// SIMATIC S7-200 project (STEP 7-Micro/WIN), CPU 224XP REL 02.01

ORGANIZATION_BLOCK MAIN:OB1
TITLE=程序注释
BEGIN
Network 2
AB=    VB135, 2
AB=    VB101, 35
AB=    VB112, 36
Network 3
AB=    VB135, 3
AB=    VB101, 35
AB=    VB126, 36
Network 5
AB<>   SMB186, 0
RCV    VB100, 0
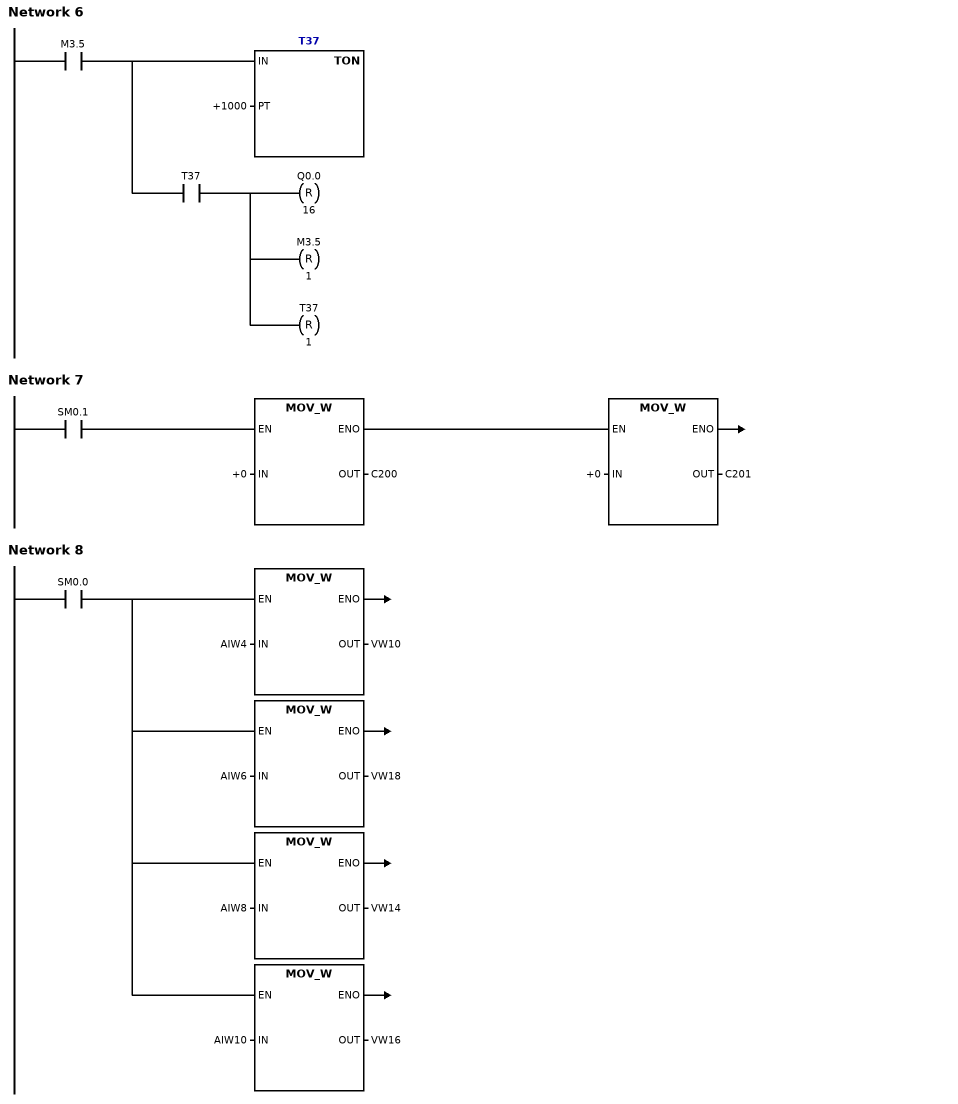
Network 6
LD     M3.5
TON    T37, +1000
A      T37
R      Q0.0, 16
R      M3.5, 1
R      T37, 1
Network 7
LD     SM0.1
MOVW   +0, C200
AENO
MOVW   +0, C201
Network 8
LD     SM0.0
MOVW   AIW4, VW10
MOVW   AIW6, VW18
MOVW   AIW8, VW14
MOVW   AIW10, VW16
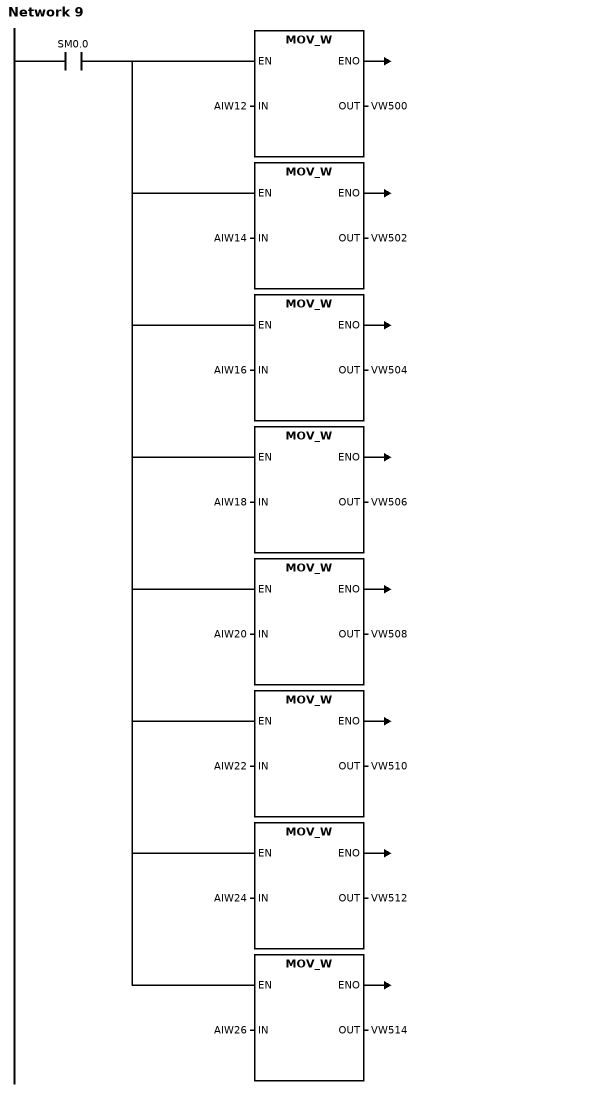
Network 9
LD     SM0.0
MOVW   AIW12, VW500
MOVW   AIW14, VW502
MOVW   AIW16, VW504
MOVW   AIW18, VW506
MOVW   AIW20, VW508
MOVW   AIW22, VW510
MOVW   AIW24, VW512
MOVW   AIW26, VW514
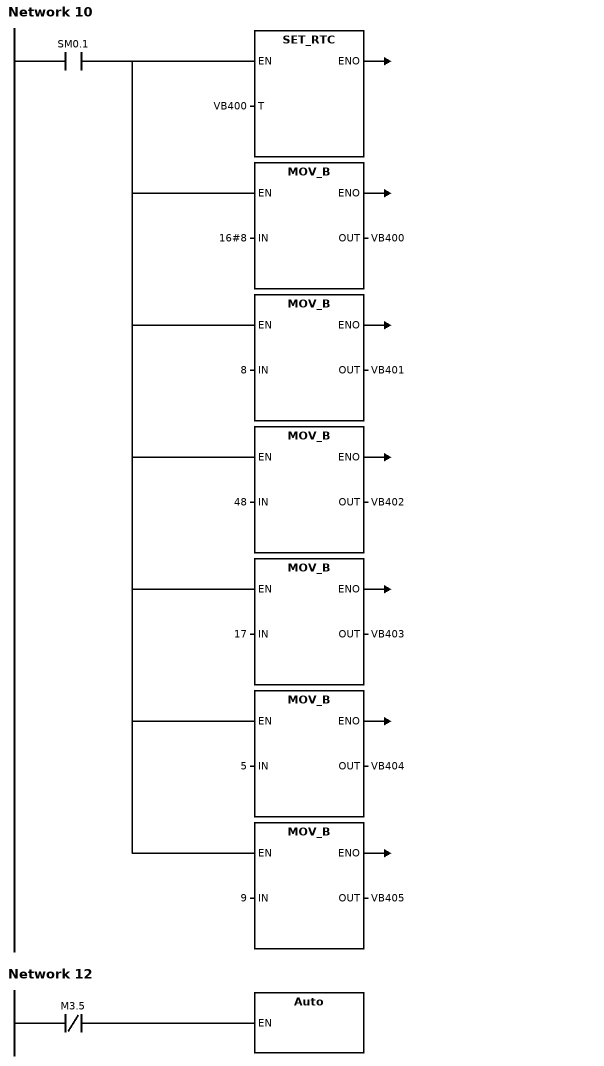
Network 10
LD     SM0.1
TODW   VB400
MOVB   16#8, VB400
MOVB   8, VB401
MOVB   48, VB402
MOVB   17, VB403
MOVB   5, VB404
MOVB   9, VB405
Network 11
LDN    I4.7
Network 12
LDN    M3.5
CALL   Auto:SBR4
Network 13
AB=    VB135, 1
AB=    VB101, 35
AB=    VB106, 36
Network 14
AB=    VB135, 5
AB=    VB101, 35
AB=    VB106, 36
S      M18.0, 1
Network 15
AB=    VB135, 6
AB=    VB101, 35
AB=    VB106, 36
S      M18.1, 1
END_ORGANIZATION_BLOCK

SUBROUTINE_BLOCK Auto:SBR4
TITLE=
BEGIN
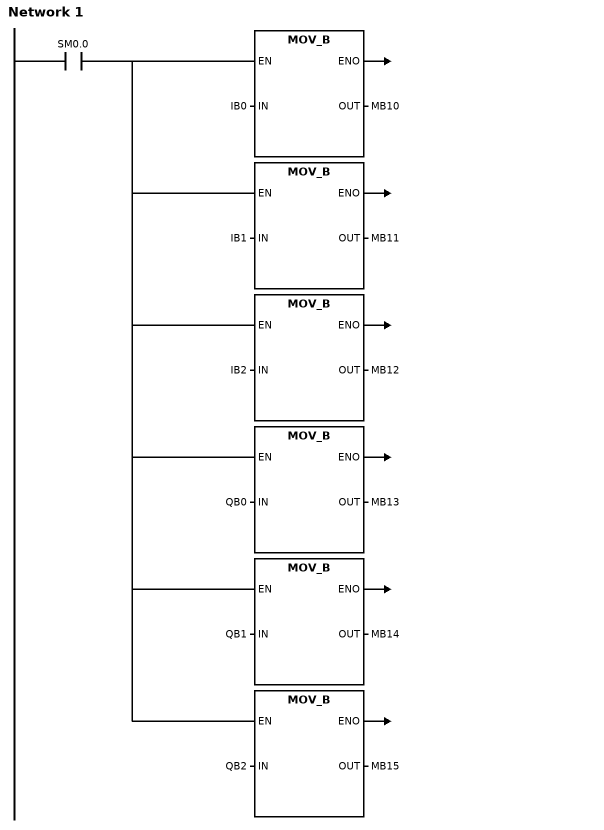
Network 1
LD     SM0.0
MOVB   IB0, MB10
MOVB   IB1, MB11
MOVB   IB2, MB12
MOVB   QB0, MB13
MOVB   QB1, MB14
MOVB   QB2, MB15
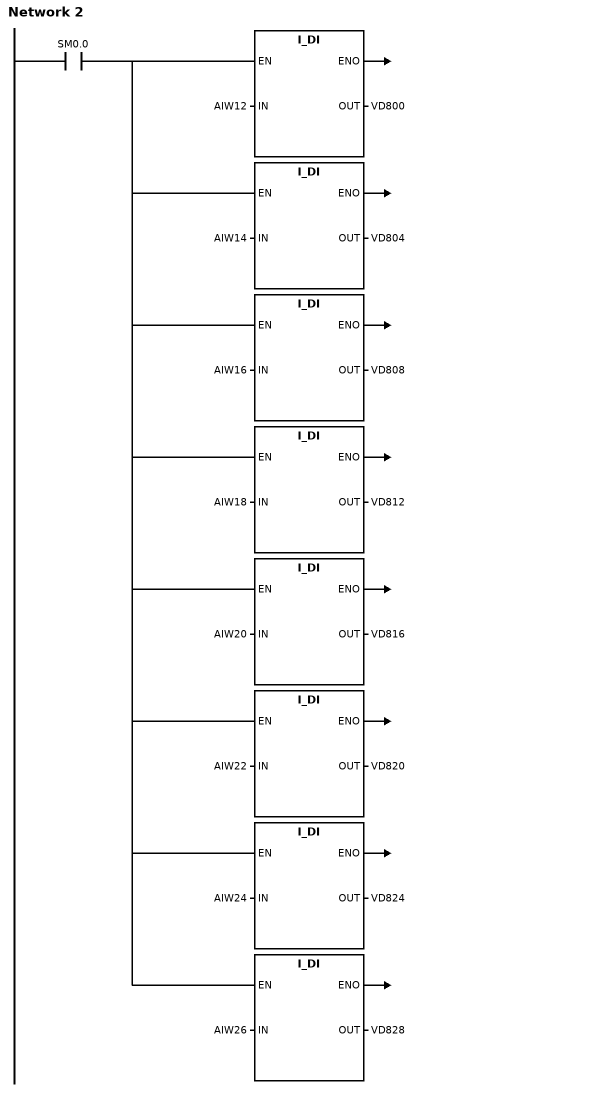
Network 2
LD     SM0.0
ITD    AIW12, VD800
ITD    AIW14, VD804
ITD    AIW16, VD808
ITD    AIW18, VD812
ITD    AIW20, VD816
ITD    AIW22, VD820
ITD    AIW24, VD824
ITD    AIW26, VD828
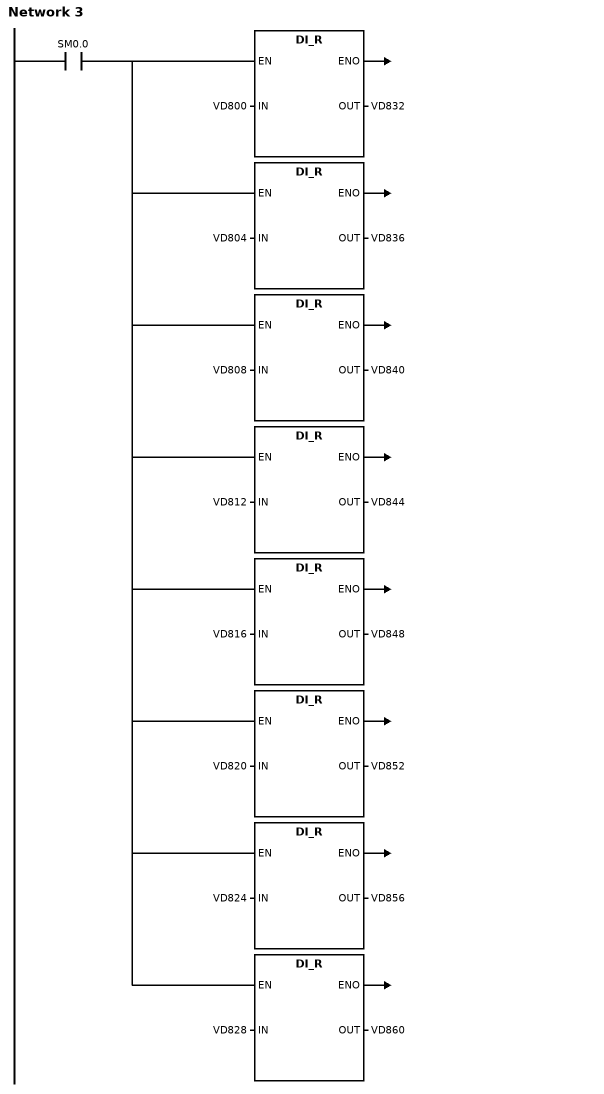
Network 3
LD     SM0.0
DTR    VD800, VD832
DTR    VD804, VD836
DTR    VD808, VD840
DTR    VD812, VD844
DTR    VD816, VD848
DTR    VD820, VD852
DTR    VD824, VD856
DTR    VD828, VD860
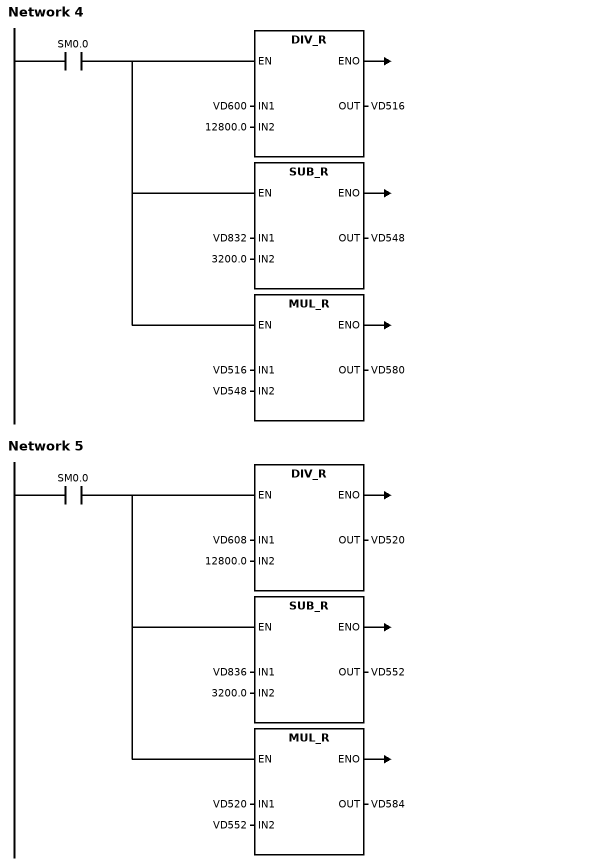
Network 4
LD     SM0.0
MOVR   VD600, VD516
/R     12800.0, VD516
MOVR   VD832, VD548
-R     3200.0, VD548
MOVR   VD516, VD580
*R     VD548, VD580
Network 5
LD     SM0.0
MOVR   VD608, VD520
/R     12800.0, VD520
MOVR   VD836, VD552
-R     3200.0, VD552
MOVR   VD520, VD584
*R     VD552, VD584
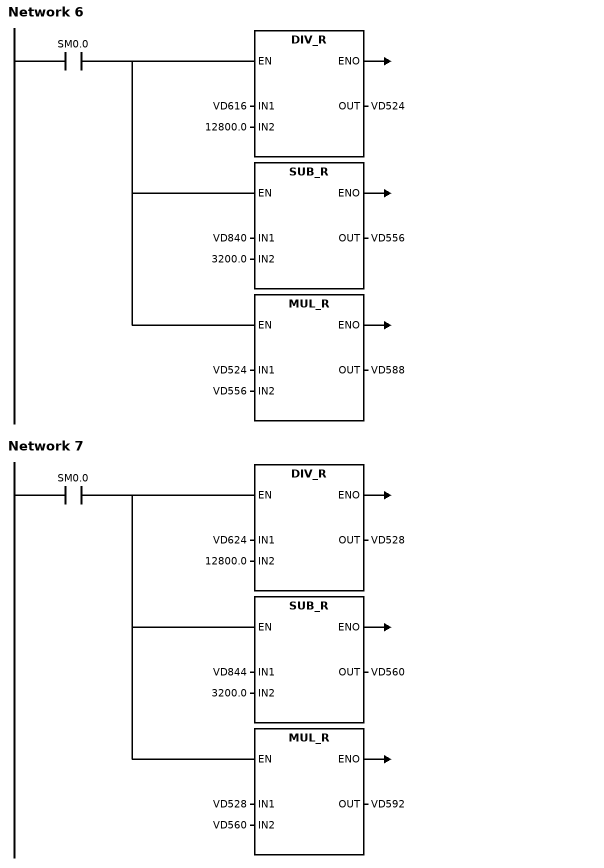
Network 6
LD     SM0.0
MOVR   VD616, VD524
/R     12800.0, VD524
MOVR   VD840, VD556
-R     3200.0, VD556
MOVR   VD524, VD588
*R     VD556, VD588
Network 7
LD     SM0.0
MOVR   VD624, VD528
/R     12800.0, VD528
MOVR   VD844, VD560
-R     3200.0, VD560
MOVR   VD528, VD592
*R     VD560, VD592
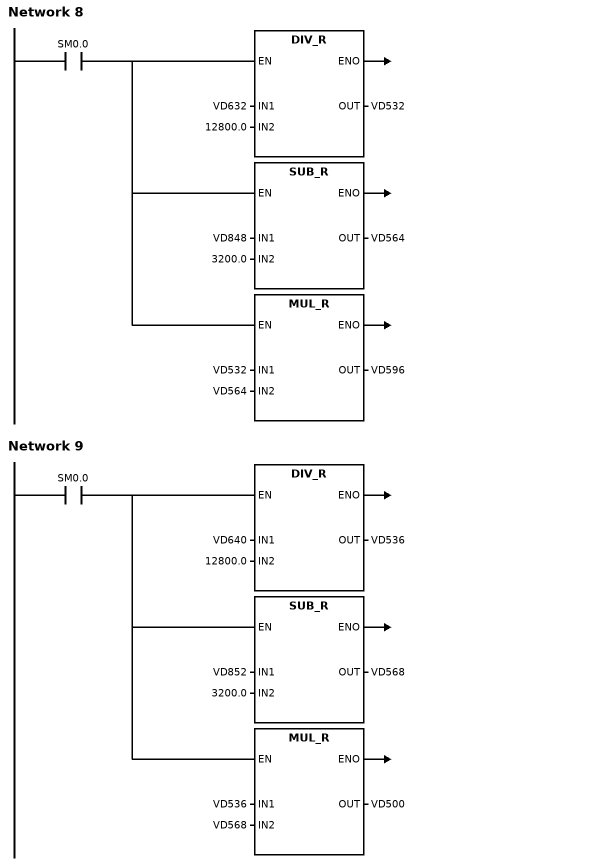
Network 8
LD     SM0.0
MOVR   VD632, VD532
/R     12800.0, VD532
MOVR   VD848, VD564
-R     3200.0, VD564
MOVR   VD532, VD596
*R     VD564, VD596
Network 9
LD     SM0.0
MOVR   VD640, VD536
/R     12800.0, VD536
MOVR   VD852, VD568
-R     3200.0, VD568
MOVR   VD536, VD500
*R     VD568, VD500
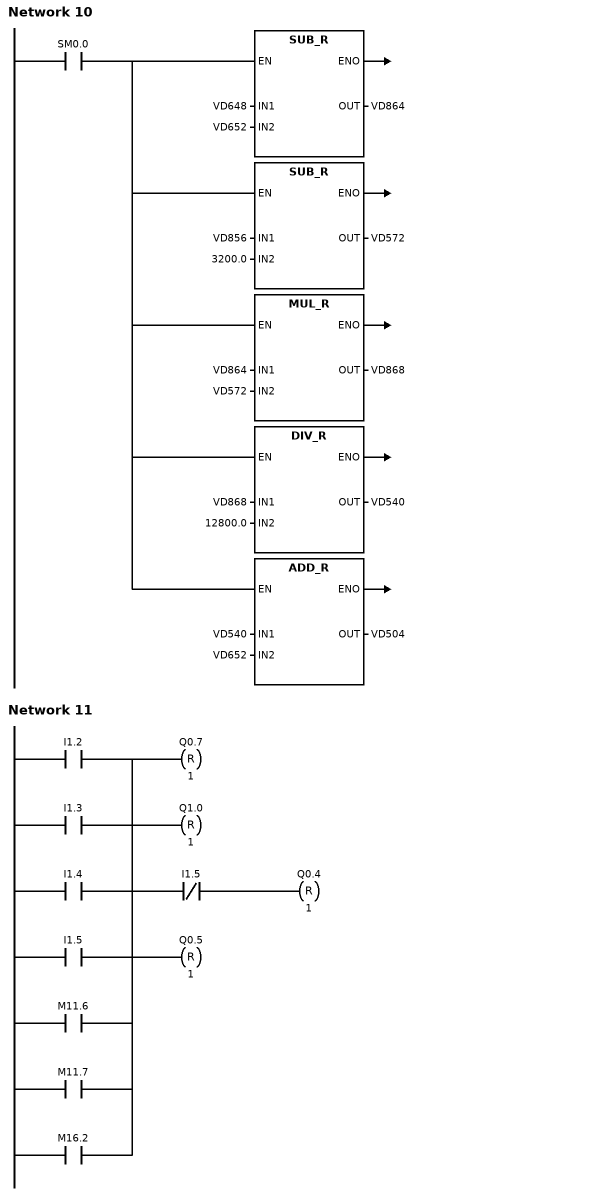
Network 10
LD     SM0.0
MOVR   VD648, VD864
-R     VD652, VD864
MOVR   VD856, VD572
-R     3200.0, VD572
MOVR   VD864, VD868
*R     VD572, VD868
MOVR   VD868, VD540
/R     12800.0, VD540
MOVR   VD540, VD504
+R     VD652, VD504
Network 11
LD     I1.2
O      I1.3
O      I1.4
O      I1.5
O      M11.6
O      M11.7
O      M16.2
LPS
R      Q0.7, 1
R      Q1.0, 1
AN     I1.5
R      Q0.4, 1
LPP
R      Q0.5, 1
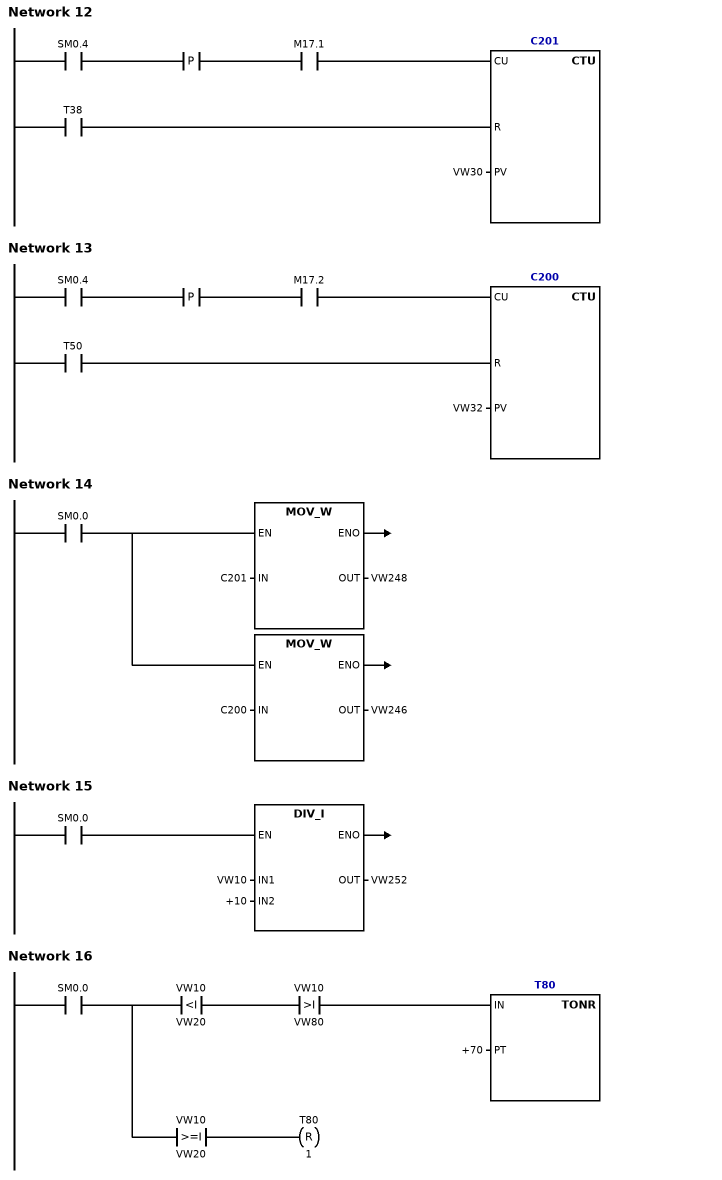
Network 12
LD     SM0.4
EU
A      M17.1
LD     T38
CTU    C201, VW30
Network 13
LD     SM0.4
EU
A      M17.2
LD     T50
CTU    C200, VW32
Network 14
LD     SM0.0
MOVW   C201, VW248
MOVW   C200, VW246
Network 15
LD     SM0.0
MOVW   VW10, VW252
/I     +10, VW252
Network 16
LD     SM0.0
LPS
AW<    VW10, VW20
AW>    VW10, VW80
TONR   T80, +70
LPP
AW>=   VW10, VW20
R      T80, 1
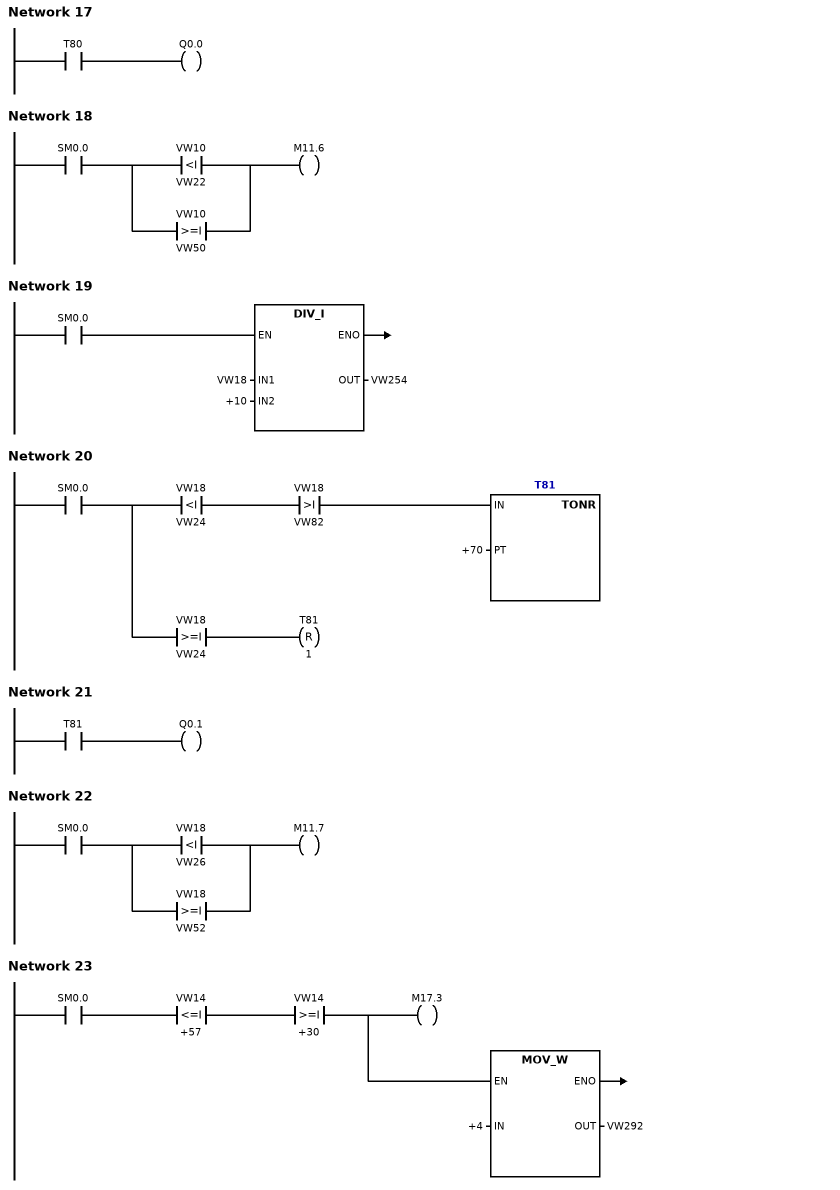
Network 17
LD     T80
=      Q0.0
Network 18
LD     SM0.0
LDW<   VW10, VW22
OW>=   VW10, VW50
ALD
=      M11.6
Network 19
LD     SM0.0
MOVW   VW18, VW254
/I     +10, VW254
Network 20
LD     SM0.0
LPS
AW<    VW18, VW24
AW>    VW18, VW82
TONR   T81, +70
LPP
AW>=   VW18, VW24
R      T81, 1
Network 21
LD     T81
=      Q0.1
Network 22
LD     SM0.0
LDW<   VW18, VW26
OW>=   VW18, VW52
ALD
=      M11.7
Network 23
LD     SM0.0
AW<=   VW14, +57
AW>=   VW14, +30
=      M17.3
MOVW   +4, VW292
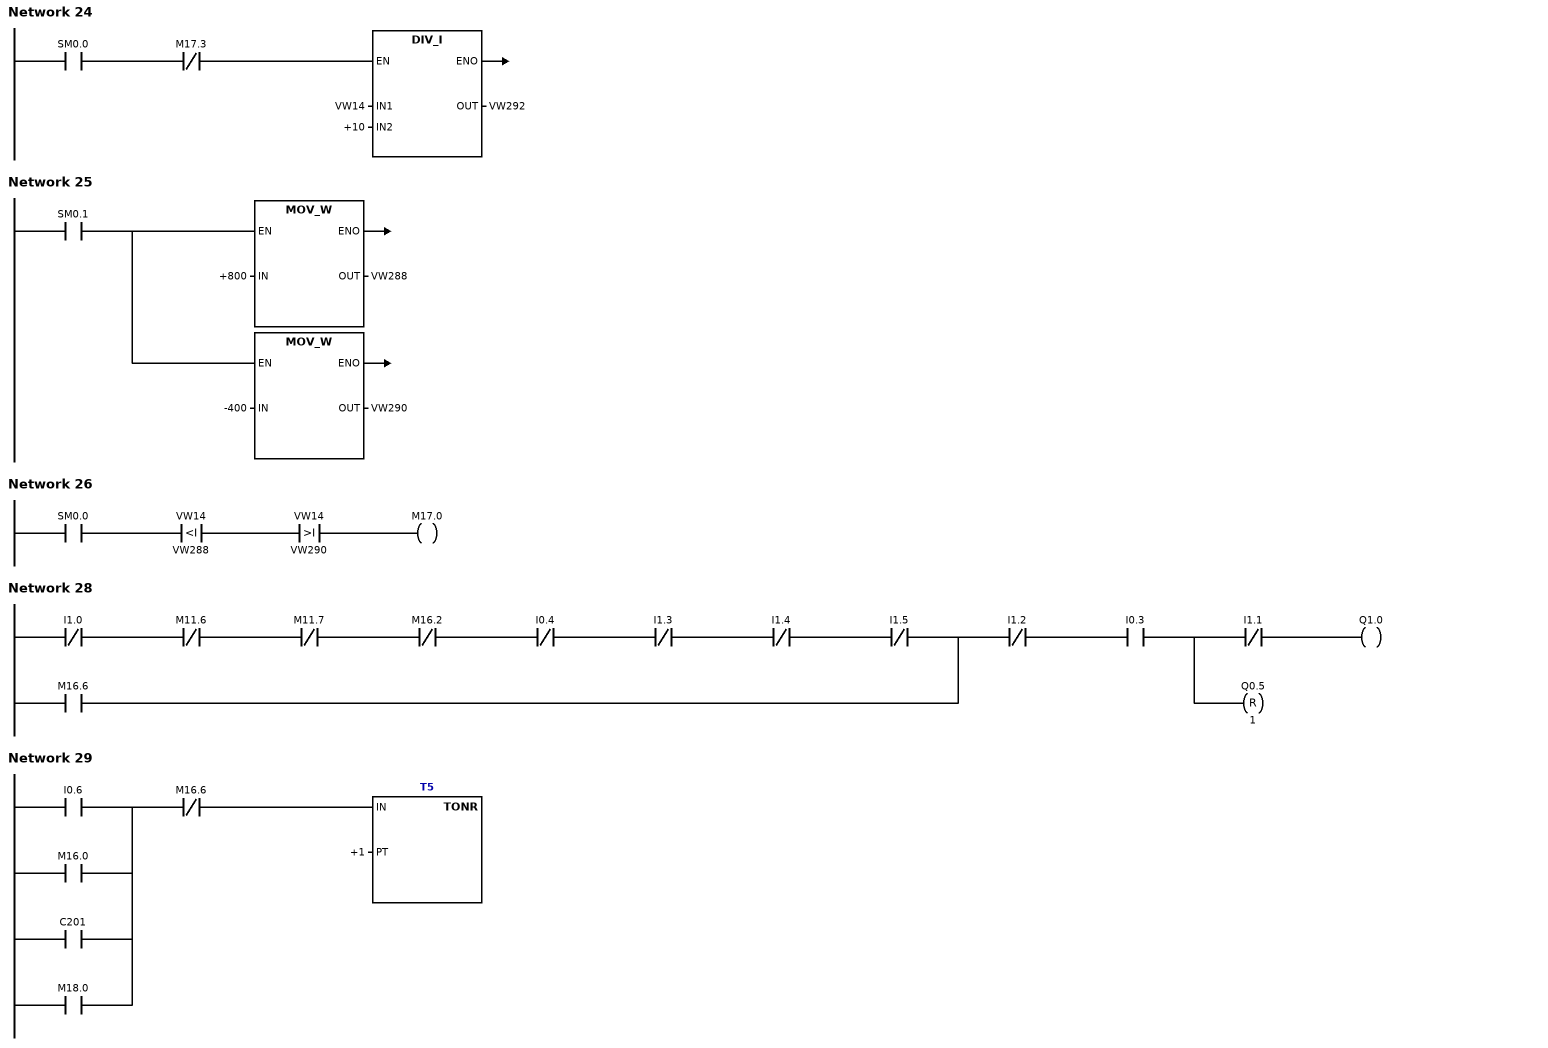
Network 24
LD     SM0.0
AN     M17.3
MOVW   VW14, VW292
/I     +10, VW292
Network 25
LD     SM0.1
MOVW   +800, VW288
MOVW   -400, VW290
Network 26
LD     SM0.0
AW<    VW14, VW288
AW>    VW14, VW290
=      M17.0
Network 28
LDN    I1.0
AN     M11.6
AN     M11.7
AN     M16.2
AN     I0.4
AN     I1.3
AN     I1.4
AN     I1.5
O      M16.6
AN     I1.2
A      I0.3
LPS
AN     I1.1
=      Q1.0
LPP
R      Q0.5, 1
Network 29
LD     I0.6
O      M16.0
O      C201
O      M18.0
AN     M16.6
TONR   T5, +1
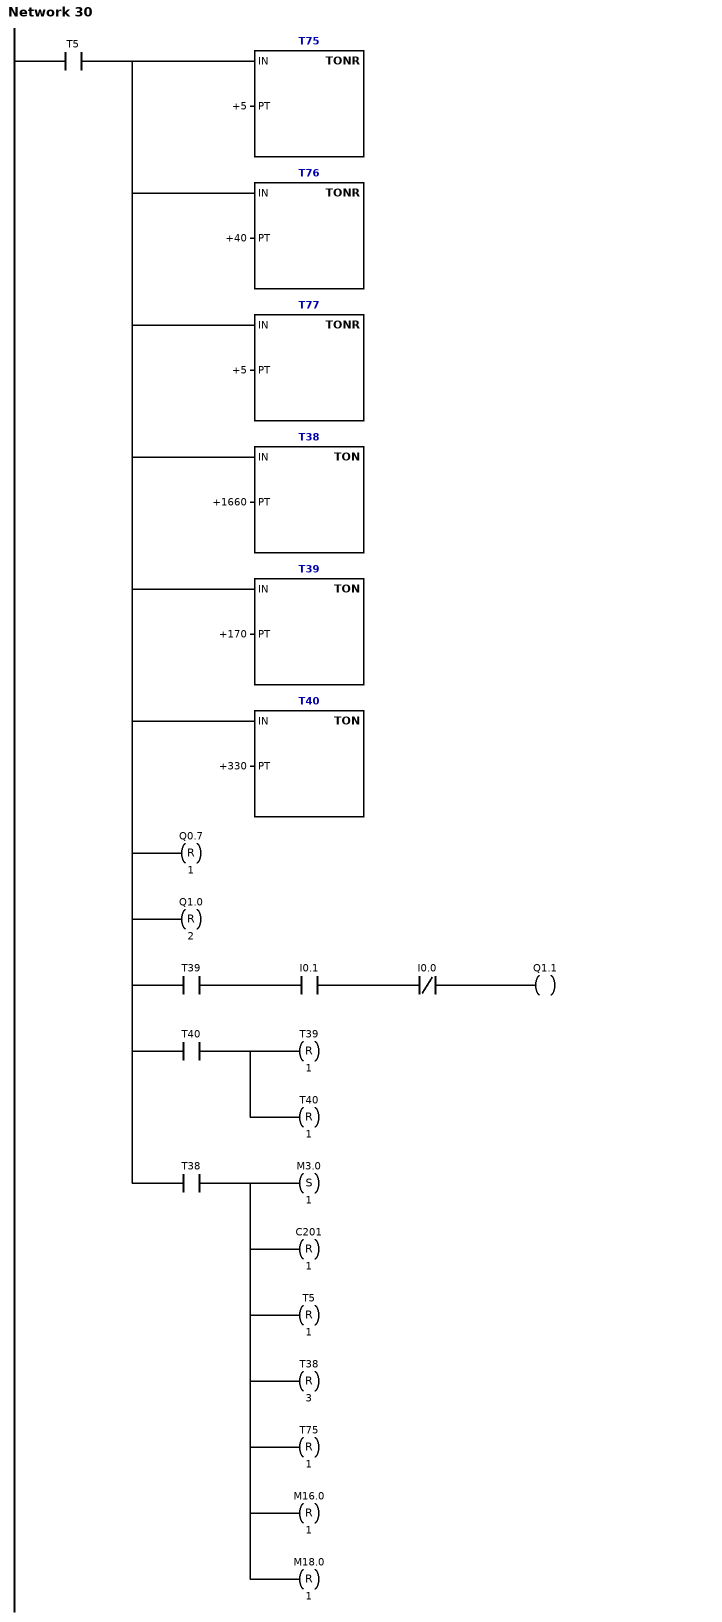
Network 30
LD     T5
LPS
TONR   T75, +5
TONR   T76, +40
TONR   T77, +5
TON    T38, +1660
TON    T39, +170
TON    T40, +330
R      Q0.7, 1
R      Q1.0, 2
A      T39
A      I0.1
AN     I0.0
=      Q1.1
LRD
A      T40
R      T39, 1
R      T40, 1
LPP
A      T38
S      M3.0, 1
R      C201, 1
R      T5, 1
R      T38, 3
R      T75, 1
R      M16.0, 1
R      M18.0, 1
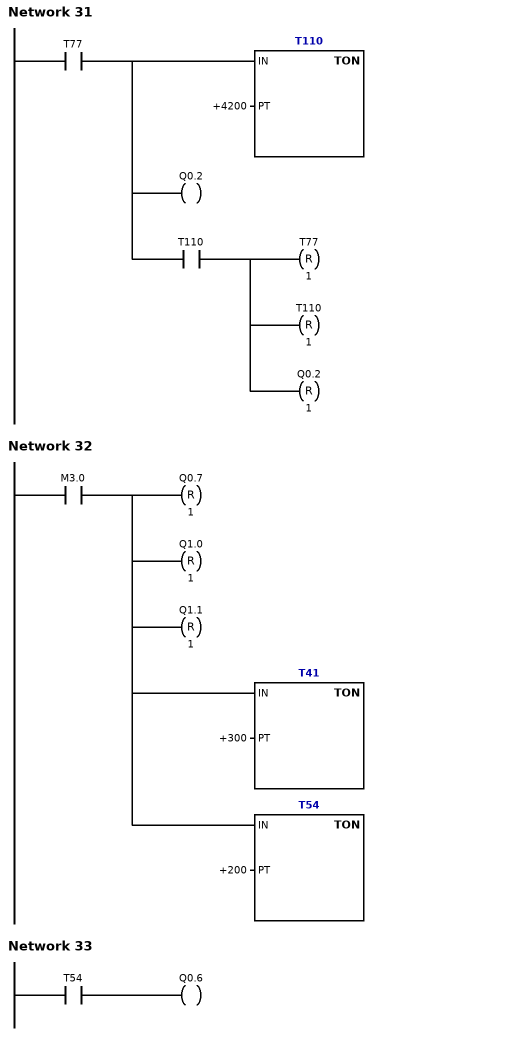
Network 31
LD     T77
TON    T110, +4200
=      Q0.2
A      T110
R      T77, 1
R      T110, 1
R      Q0.2, 1
Network 32
LD     M3.0
R      Q0.7, 1
R      Q1.0, 1
R      Q1.1, 1
TON    T41, +300
TON    T54, +200
Network 33
LD     T54
=      Q0.6
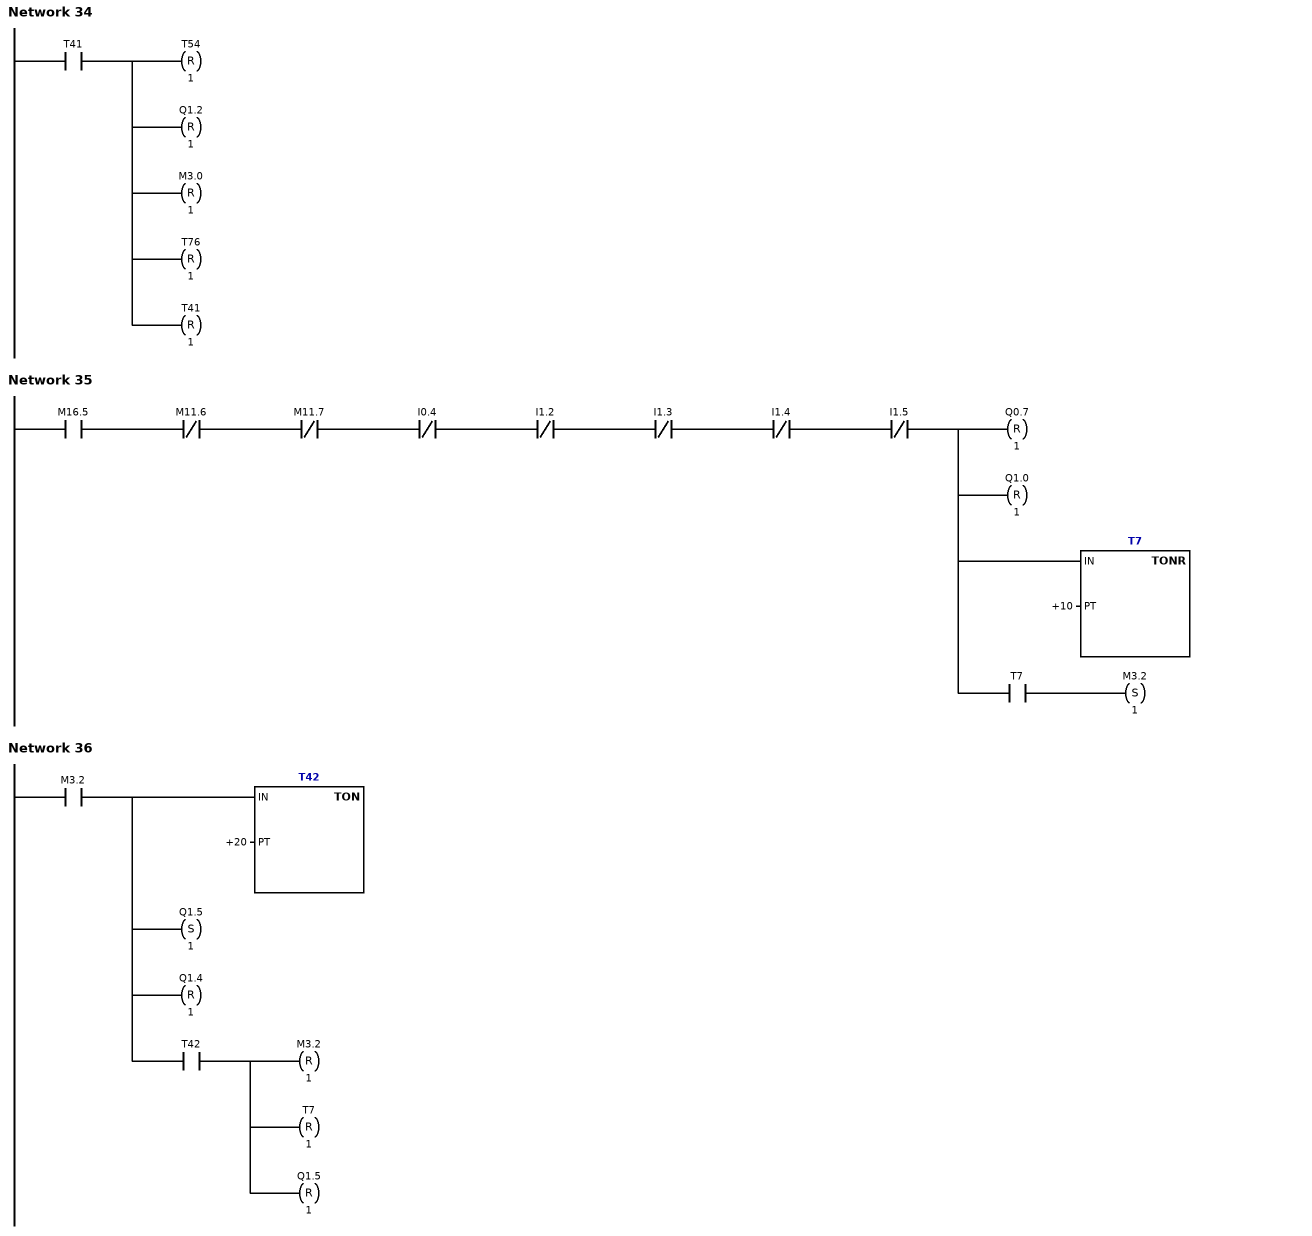
Network 34
LD     T41
R      T54, 1
R      Q1.2, 1
R      M3.0, 1
R      T76, 1
R      T41, 1
Network 35
LD     M16.5
AN     M11.6
AN     M11.7
AN     I0.4
AN     I1.2
AN     I1.3
AN     I1.4
AN     I1.5
R      Q0.7, 1
R      Q1.0, 1
TONR   T7, +10
A      T7
S      M3.2, 1
Network 36
LD     M3.2
TON    T42, +20
S      Q1.5, 1
R      Q1.4, 1
A      T42
R      M3.2, 1
R      T7, 1
R      Q1.5, 1
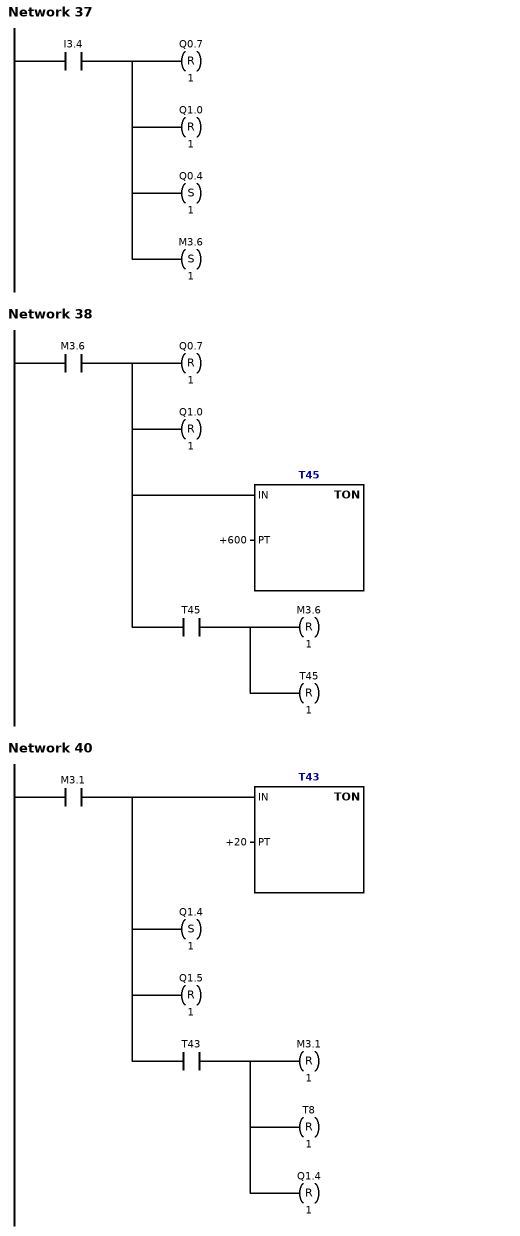
Network 37
LD     I3.4
R      Q0.7, 1
R      Q1.0, 1
S      Q0.4, 1
S      M3.6, 1
Network 38
LD     M3.6
R      Q0.7, 1
R      Q1.0, 1
TON    T45, +600
A      T45
R      M3.6, 1
R      T45, 1
Network 39
AN     M11.6
AN     M11.7
AN     I1.0
AN     I1.2
AN     I1.3
AN     I1.4
AN     I1.5
R      Q0.7, 1
R      Q1.0, 1
TONR   T8, +10
A      T8
S      M3.1, 1
Network 40
LD     M3.1
TON    T43, +20
S      Q1.4, 1
R      Q1.5, 1
A      T43
R      M3.1, 1
R      T8, 1
R      Q1.4, 1
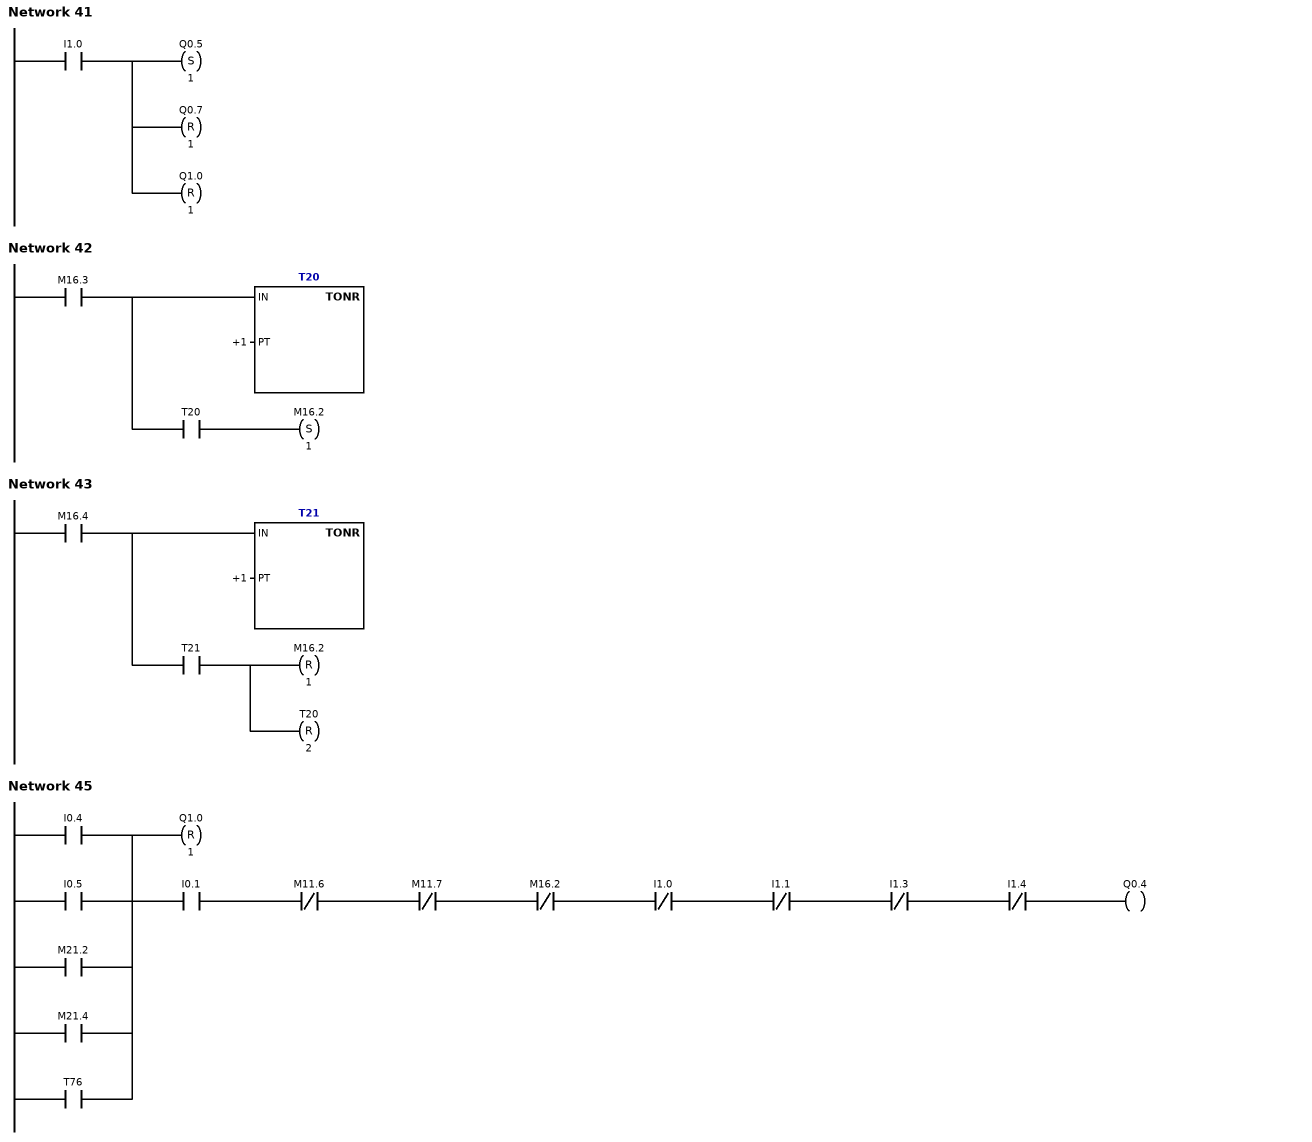
Network 41
LD     I1.0
S      Q0.5, 1
R      Q0.7, 1
R      Q1.0, 1
Network 42
LD     M16.3
TONR   T20, +1
A      T20
S      M16.2, 1
Network 43
LD     M16.4
TONR   T21, +1
A      T21
R      M16.2, 1
R      T20, 2
Network 45
LD     I0.4
O      I0.5
O      M21.2
O      M21.4
O      T76
R      Q1.0, 1
A      I0.1
AN     M11.6
AN     M11.7
AN     M16.2
AN     I1.0
AN     I1.1
AN     I1.3
AN     I1.4
=      Q0.4
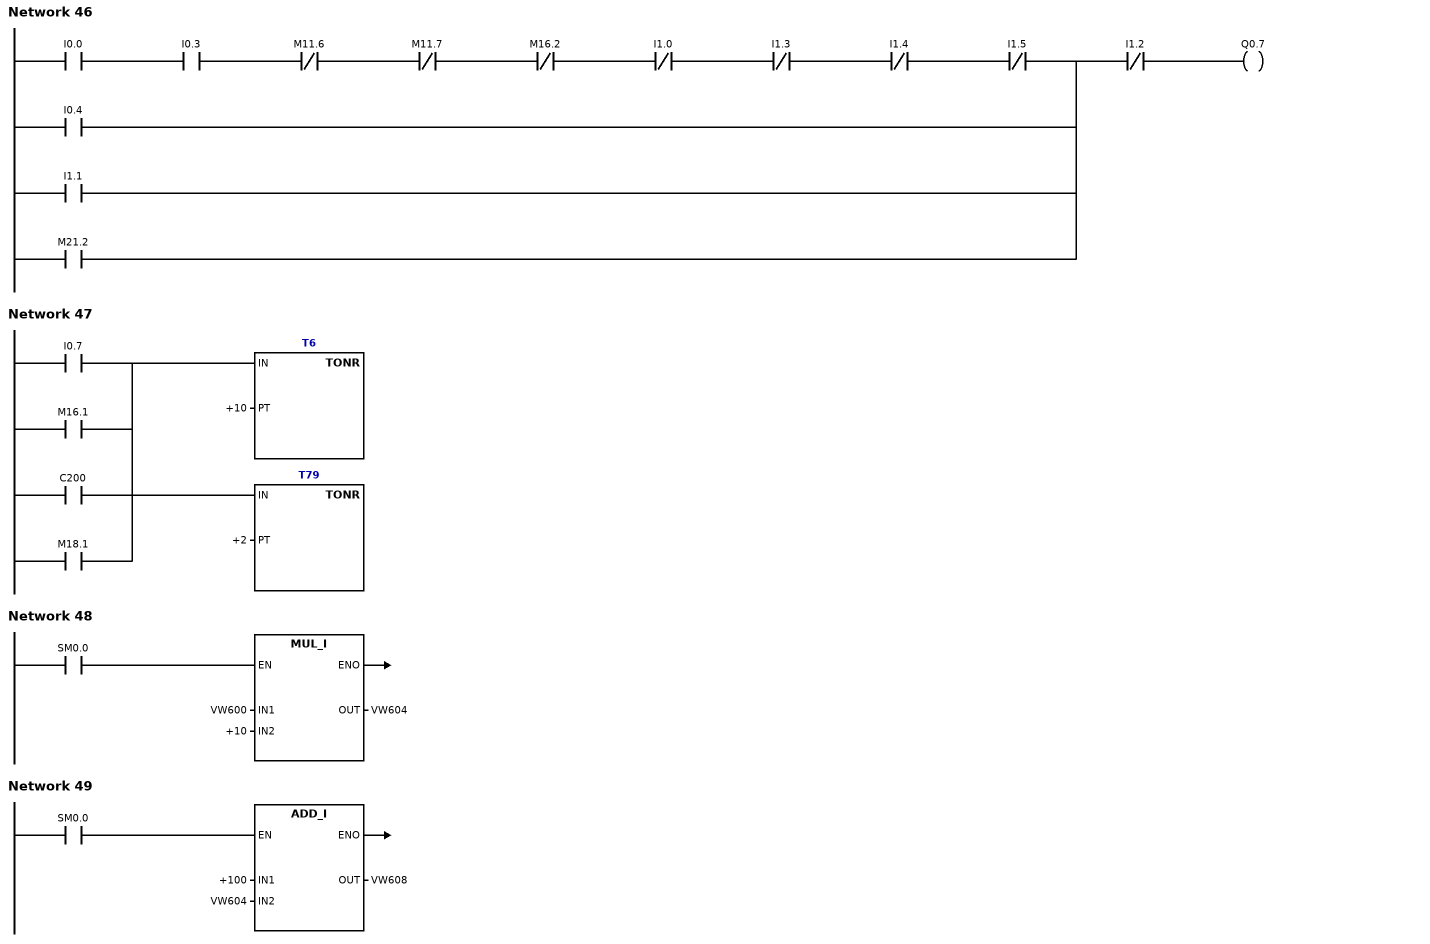
Network 46
LD     I0.0
A      I0.3
AN     M11.6
AN     M11.7
AN     M16.2
AN     I1.0
AN     I1.3
AN     I1.4
AN     I1.5
O      I0.4
O      I1.1
O      M21.2
AN     I1.2
=      Q0.7
Network 47
LD     I0.7
O      M16.1
O      C200
O      M18.1
TONR   T6, +10
TONR   T79, +2
Network 48
LD     SM0.0
MOVW   VW600, VW604
*I     +10, VW604
Network 49
LD     SM0.0
MOVW   +100, VW608
+I     VW604, VW608
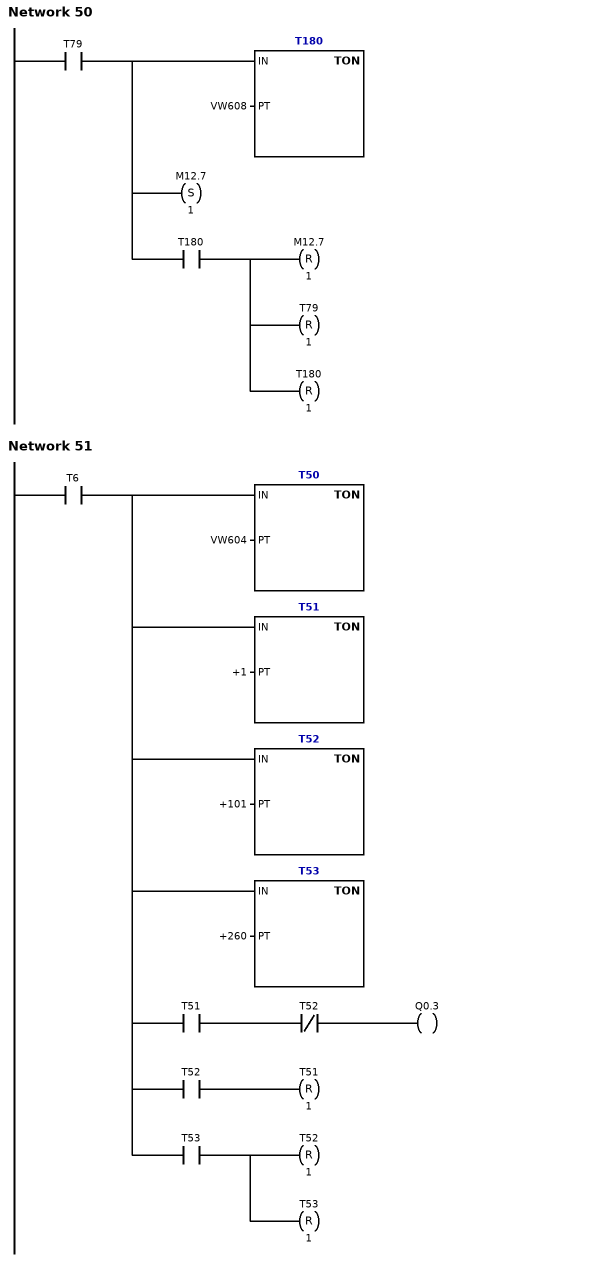
Network 50
LD     T79
TON    T180, VW608
S      M12.7, 1
A      T180
R      M12.7, 1
R      T79, 1
R      T180, 1
Network 51
LD     T6
LPS
TON    T50, VW604
TON    T51, +1
TON    T52, +101
TON    T53, +260
A      T51
AN     T52
=      Q0.3
LRD
A      T52
R      T51, 1
LPP
A      T53
R      T52, 1
R      T53, 1
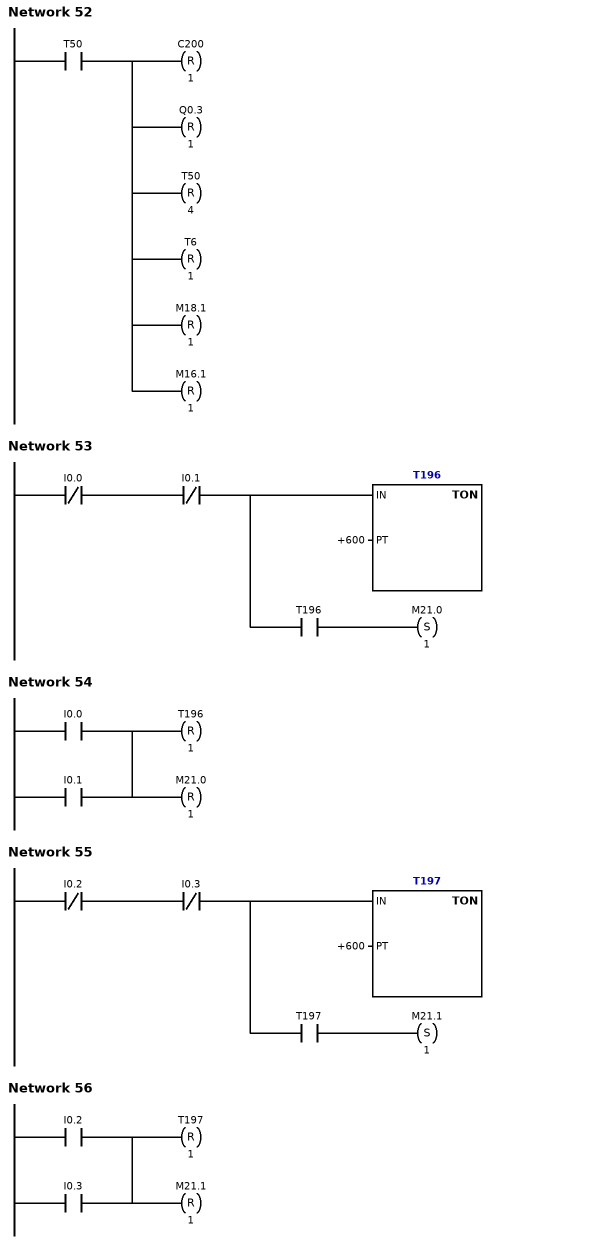
Network 52
LD     T50
R      C200, 1
R      Q0.3, 1
R      T50, 4
R      T6, 1
R      M18.1, 1
R      M16.1, 1
Network 53
LDN    I0.0
AN     I0.1
TON    T196, +600
A      T196
S      M21.0, 1
Network 54
LD     I0.0
O      I0.1
R      T196, 1
R      M21.0, 1
Network 55
LDN    I0.2
AN     I0.3
TON    T197, +600
A      T197
S      M21.1, 1
Network 56
LD     I0.2
O      I0.3
R      T197, 1
R      M21.1, 1
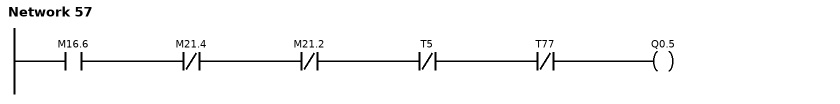
Network 57
LD     M16.6
AN     M21.4
AN     M21.2
AN     T5
AN     T77
=      Q0.5
END_SUBROUTINE_BLOCK

SUBROUTINE_BLOCK AutoRead:SBR5
TITLE=
BEGIN
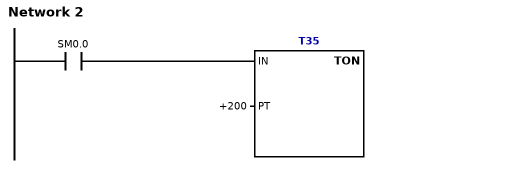
Network 2
LD     SM0.0
TON    T35, +200
Network 3
LD     T35
MOVB   58, VB300
MOVB   56, VB301
MOVB   56, VB302
MOVB   56, VB303
MOVB   56, VB304
MOVB   56, VB305
MOVB   56, VB306
MOVB   56, VB307
MOVB   48, VB308
MOVB   48, VB309
MOVB   48, VB310
MOVB   48, VB311
MOVB   52, VB312
MOVB   51, VB313
MOVB   51, VB314
MOVB   52, VB315
MOVB   50, VB316
MOVW   AIW0, VW317
MOVW   AIW2, VW319
MOVW   AIW4, VW321
MOVW   AIW6, VW323
MOVW   AIW8, VW325
MOVW   AIW10, VW327
MOVW   AIW12, VW329
MOVW   AIW14, VW331
MOVW   AIW16, VW333
MOVW   AIW18, VW335
MOVW   AIW20, VW337
MOVW   AIW22, VW339
MOVW   AIW24, VW341
MOVW   AIW26, VW343
MOVW   VW20, VW345
MOVW   VW24, VW347
MOVW   VW32, VW349
MOVW   VW30, VW351
MOVB   IB0, VB353
MOVB   IB1, VB354
MOVB   IB2, VB355
MOVB   QB0, VB356
MOVB   QB1, VB357
MOVB   QB2, VB358
END_SUBROUTINE_BLOCK

// (further data pages could not be read)
